Staubli VAL3: create_cylinder.pgx

public program create_cylinder(point x_pOrigin, num x_nRadius, num x_nDistanceZ)
begin
  //
  // build the Cylinder
  //
  if setFrame(x_pOrigin,compose(x_pOrigin,world,{x_nRadius,0,0,0,0,0}),compose(x_pOrigin,world,{0,x_nRadius,0,0,0,0}),fCylinder)==0
    bCreate_cylind=true
  else
    bCreate_cylind=false
  endIf
  // copy all
  nRadius_cyl=x_nRadius
  nDistanceZ_cyl=x_nDistanceZ
  pOrigin_cylind.trsf=position(x_pOrigin,world)
end
